// TwinCAT 3 PLC project CLOCK
// ProgramVersion: 3.1.4022.2
// libraries:
//   Tc2_EtherCAT, * (Beckhoff Automation GmbH)
//   Tc2_Standard, * (Beckhoff Automation GmbH)
//   Tc2_System, * (Beckhoff Automation GmbH)
//   Tc2_Utilities, * (Beckhoff Automation GmbH)
//   Tc3_Module, * (Beckhoff Automation GmbH)
// project tree:
//   / PlcTask.TcTTO
//   POUs/ MAIN.TcPOU
// real-time tasks:
//   TASK Plc_Task_CLOCK: cycle T#1ms, priority 20, ADS port 350
//   TASK Plc_Task_SYNC: cycle T#10ms, priority 21, ADS port 351
// motion (NC):
//   TASK NC-Task 1 SAF: cycle T#2ms, priority 4, ADS port 501
//   TASK NC-Task 1 SVB: cycle T#10ms, priority 8, ADS port 511
//   AXIS SyncMaster (id 1)
//     General: UnitName=°, UnitFlags=#x00000004
//     Velo: Maximum=5750
//     OtherSettings: AllowMotionCmdToSlave=true
//     encoder EncType=1
//     drive DrvType=5
//       Analog: VeloReferenz=6000, ScaleFactorActTorque=0.1
//       TimeComp: TaskDelayCycles=1
//     controller CtrType=1
//       CtrPara: PriorControlFactor=1
//         Observer: BandWidth=20
//   AXIS SyncSlave (id 2)
//     General: UnitName=°, UnitFlags=#x00000004
//     Velo: Maximum=10000
//     OtherSettings: AllowMotionCmdToSlave=true
//     encoder EncType=1
//     drive DrvType=5
//       Analog: VeloReferenz=10000, ScaleFactorActTorque=0.1
//     controller CtrType=1
//       CtrPara: PriorControlFactor=1
//         Observer: BandWidth=20
// variable links:
//   CLOCK Instance <-> SYNC/SYNC Instance
//     PlcTask Outputs/MAIN.tPulse <-> Plc_Task_SYNC Inputs/MAIN.tPulse
//   SYNC Instance <-> NC-Task 1 SAF/Axes/SyncMaster
//     Plc_Task_SYNC Inputs/MAIN.SyncMaster.NcToPlc <-> Outputs/ToPlc
//     Plc_Task_SYNC Outputs/MAIN.SyncMaster.PlcToNc <-> Inputs/FromPlc
//   SYNC Instance <-> NC-Task 1 SAF/Axes/SyncSlave
//     Plc_Task_SYNC Inputs/MAIN.SyncSlave.NcToPlc <-> Outputs/ToPlc
//     Plc_Task_SYNC Outputs/MAIN.SyncSlave.PlcToNc <-> Inputs/FromPlc

CONFIGURATION CLOCK
    RESOURCE PLC ON TwinCAT3
        TASK PlcTask(INTERVAL := T#1ms, PRIORITY := 20);
        PROGRAM MAIN WITH PlcTask : MAIN;
    END_RESOURCE
END_CONFIGURATION

// ---- POUs/MAIN.TcPOU
PROGRAM MAIN
VAR
	iFreq : INT := 14;
	tPeriod : TIME;
	
	tPulse AT %Q*: T_DCTIME64;
	
	tDelta : T_DCTIME64;
	tsDelta : DCTIMESTRUCT;
	iJitter : DINT; // Microseconds of jitter
	
	iState : UINT;
	
	fbTimer : TON;
END_VAR

CASE iState OF
	0:
		// Calculate the period
		tPeriod := T#1S/iFreq;
		fbTimer.PT := tPeriod - T#3MS;
		
		// Start the timer
		fbTimer.IN:=TRUE;

		iState := 1;
		
	1:
		// Wait for timer to complete
		IF fbTimer.Q THEN
			tDelta := tPulse;
			
			// Get the DC time
			tPulse := F_GetCurDcTaskTime64();
			
			tDelta := tPulse - tDelta;
			
			tsDelta := DCTIME64_TO_DCTIMESTRUCT(tDelta);
			
			iJitter := - TIME_TO_DINT(tPeriod);
			iJitter := iJitter + tsDelta.wSecond * 1000;
			iJitter := iJitter + tsDelta.wMilliseconds;
			iJitter := iJitter * 1000 + tsDelta.wMicroseconds;
			
			iState:= 2;
		END_IF
		
	2:
		// Reset the timer
		fbTimer.IN := FALSE;
		
		iState := 0;
END_CASE

fbTimer();

END_PROGRAM
